// TIA Portal V19 export
TYPE "lexchangetray_typeroller_signalTM_ControlNode_1"
// Type: lexchangetray_typeroller_signalTM_Simulation_1
// Type: lexchangetray_typeroller_signalTM_Monitor_1
// Type: lexchangetray_typeroller_signalTM_Cmd_1
// stored: Access Published
   STRUCT
      cmd : "lexchangetray_typeroller_signalTM_Cmd_1";
      monitor { S7_SetPoint := 'True'} : "lexchangetray_typeroller_signalTM_Monitor_1";
      sim { S7_SetPoint := 'True'} : "lexchangetray_typeroller_signalTM_Simulation_1";
   END_STRUCT;
END_TYPE
